(* Logix 5000 project; controller RSL5k_18_Template_noLib Emulate 5570 rev 32.11; software revision 32.02; part 4 of 16 *)
(* tags used below, declared in another part *)
   Cfg_AllowDisable : BOOL;   // 1=Allow Maintenance to Disable this Alarm
   PCmd_Reset : BOOL;   // Program Command to Reset latched alarm
   PCmd_Ack : BOOL;   // Program Command to Acknowledge alarm
   PCmd_Suppress : BOOL;   // Program Command to Suppress by Design (inhibits new alarm)
   PCmd_Unsuppress : BOOL;   // Program Command to Unsuppress (allows new alarm)
   PCmd_Unshelve : BOOL;   // Program Command to Unshelve (e.g., on shift change)
   Shelved : ALIAS FOR Com_AE.3;   // 1=Alarm has been Shelved by Operator (inhibits new alarm)
   Suppressed : ALIAS FOR Com_AE.6;   // 1=Alarm has been Suppressed by Program (inhibits new alarm)
   Disabled : ALIAS FOR Com_AE.9;   // 1=Alarm has been Disabled by Maintanance (inhibits new alarm)
   P_Alarm : BOOL;   // Unique Parameter Name for auto - discovery
   Wrk_Suppressed : BOOL;   // Internal Alarm Suppressed Status
   Com_AE : INT;   // Communication with HMI / Alarm/Event Server (see bit descriptions)
   OCmd_Unshelve : BOOL;   // Operator Command to Unshelve alarm (allows new alarm)
   OCmd_Shelve : BOOL;   // Operator Command to Shelve Alarm (inhibits new alarm)
   OCmd_Ack : BOOL;   // Operator Command to Acknowledge alarm
   OCmd_Reset : BOOL;   // Operator Command to Reset latched alarm
   MCmd_Enable : BOOL;   // Maintenance Command to Enable alarm (allows new alarm)
   MCmd_Disable : BOOL;   // Maintenance Command to Disable alarm (inhibits new alarm)
(* P_Alarm, continued *)

ROUTINE Prescan   (* ladder *)
// Clear "lurking" Commands
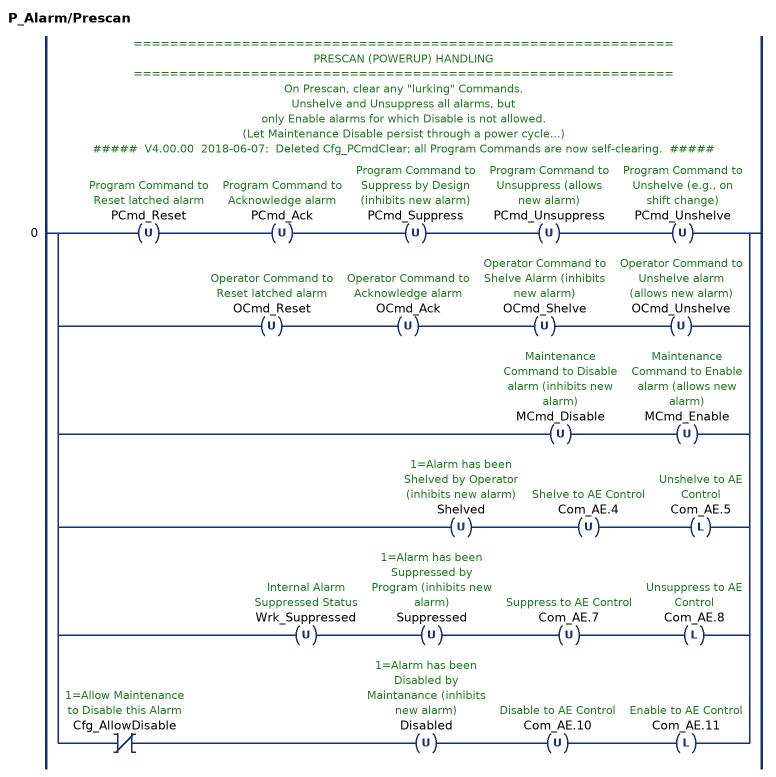
   // ============================================================
   // PRESCAN (POWERUP) HANDLING
   // ============================================================
   // On Prescan, clear any "lurking" Commands.
   // Unshelve and Unsuppress all alarms, but
   // only Enable alarms for which Disable is not allowed.
   // (Let Maintenance Disable persist through a power cycle...)
   // #####  V4.00.00  2018-06-07:  Deleted Cfg_PCmdClear; all Program Commands are now self-clearing.  #####
   0: [OTU(PCmd_Reset) OTU(PCmd_Ack) OTU(PCmd_Suppress) OTU(PCmd_Unsuppress) OTU(PCmd_Unshelve) ,OTU(OCmd_Reset) OTU(OCmd_Ack) OTU(OCmd_Shelve) OTU(OCmd_Unshelve) ,OTU(MCmd_Disable) OTU(MCmd_Enable) ,OTU(Shelved) OTU(Com_AE.4) OTL(Com_AE.5) ,OTU(Wrk_Suppressed) OTU(Suppressed) OTU(Com_AE.7) OTL(Com_AE.8) ,XIO(Cfg_AllowDisable) OTU(Disabled) OTU(Com_AE.10) OTL(Com_AE.11) ];
END_ROUTINE
END_ADD_ON_INSTRUCTION

ADD_ON_INSTRUCTION P_CmdSrc   (* revision 4.10 .01 Release, vendor Rockwell Automation, ExecutePrescan, ExecuteEnableInFalse *)
// Command Source
// Revision note:
// See Instruction Help for a summary of changes, and see 4.10 Release Notes for details.
// Help:
// Copyright © Rockwell Automation, Inc.  All Rights Reserved.
// This instruction provides selection of Command Source for a Device-
// level object  (from highest priority to lowest):
// * Not Initialized
// * Hand (hardwired control, not controllable from I/O)
// * POoS (Programmed Out of Service) (EnableIn is false)
// * MOoS (Maintenance Out of Service)
// * Maint (Maintenance)
// * Ovrd (Override) (typically used for process overrides)
// * External (e.g.: local/field devices or upstream SCADA)
// * Prog (Program) (automated control, and default if Cfg_ProgDefault = 1)
// * Oper (Operator (manual control, and default if Cfg_ProgDefault = 0)
// (Program and Operator have the same priority.)
// The current command source is shown with individual Status bits
// and also a bit field (Sts_bSrc) and an enumeration (Sts_eSrc).
// When EnableIn is false, all source acquire/release and lock/unlock
// Commands are processed "behind the scenes", but the source
// "Program Out of Service" (POoS) is selected.  When EnableIn
// becomes true, the source selection takes into account the
// Commands received -- in other words, the command source
// becomes the one that would have been in effect had the EnableIn
// False / Out of Service condition never occurred.
// SUMMARY OF CHANGES FROM PREVIOUS VERSION (4.10.00)
// See 4.10 Release Notes for details.
// * Added clear of internal "Ext" latch if Ext does not exist.
// SUMMARY OF CHANGES FROM PREVIOUS VERSION (4.00.01)
// See 4.10 Release Notes for details.
// * Added XCmd_Acq, XCmd_Rel, Cfg_ExtAcqAsLevel, removed Inp_Ext.
// * Added XRdy_Acq, XRdy_Rel so XCmd_Acq, XCmd_Rel can be used on HMI.
// * Corrected parameter external access.
// SUMMARY OF CHANGES FROM PREVIOUS VERSION (4.00.00)
// See 4.00 Release Notes for details.
// Minor change to initialization, handling of level commands in EnableInFalse.
// SUMMARY OF CHANGES FROM PREVIOUS VERSION (P_Mode V3.5-01)
// See 4.00 Release Notes for details.
// * Derived from P_Mode V3.5-01. P_Mode version history archived.
// * Added Out of Service (OoS), External (Ext); removed "NoMode"
// * Added configuration for sources to exist, commands for "opposite" source.
// * Aligned ready bit naming with command bit names.
VAR_INPUT
   Inp_Hand : BOOL; {visible}   // 1=Acquire Hand (typ. hardwired local), 0=Release Hand
   Inp_Ovrd : BOOL; {visible}   // 1=Acquire Override (higher priority program logic), 0=Release Override
   Inp_ExtInh : BOOL; {visible}   // 1=Inhibit External Acquisition, 0=Allow External Acquisition
   Cfg_HasOper : BOOL := 1;   // 1=Operator (unlocked) exists, can be selected
   Cfg_HasOperLocked : BOOL := 1;   // 1=Operator Locked exists, can be selected
   Cfg_HasProg : BOOL := 1;   // 1=Program (unlocked) exists, can be selected
   Cfg_HasProgLocked : BOOL := 1;   // 1=Program Locked exists, can be selected
   Cfg_HasExt : BOOL;   // 1=External exists, can be selected
   Cfg_HasMaint : BOOL := 1;   // 1=Maintenance exists, can be selected
   Cfg_HasMOoS : BOOL := 1;   // 1=Maintenance Out of Service exists, can be selected
   Cfg_OvrdOverLock : BOOL := 1;   // 1=Override supersedes Prog/Oper Lock, 0=don't override Lock
   Cfg_ExtOverLock : BOOL;   // 1=External supersedes Prog/Oper Lock, 0=don't override Lock
   Cfg_ProgPwrUp : BOOL;   // 1=Power Up to Prog, 0=Power Up to Oper
   Cfg_ProgNormal : BOOL;   // Normal Source: 1=Program if no requests; 0=Operator if no requests
   Cfg_PCmdPriority : BOOL;   // Command Priority: 1=Program Cmds Win; 0=Operator Cmds Win
   Cfg_PCmdProgAsLevel : BOOL;   // 1=PCmd_Prog used as a Level (1=Prog, 0=Oper)
   Cfg_PCmdLockAsLevel : BOOL;   // 1=PCmd_Lock used as a Level (1=Lock, 0=Unlock)
   Cfg_ExtAcqAsLevel : BOOL;   // 1=XCmd_Acq used as Level (1=Acq, 0=Rel)
   PCmd_Oper : BOOL;   // Program Command to select Operator (Prog to Oper)
   PCmd_Prog : BOOL;   // Program Command to select Program (Oper to Prog)
   PCmd_Lock : BOOL;   // Program Command to Lock Program (disallow Operator)
   PCmd_Unlock : BOOL;   // Program Command to Unlock Program (allow Oper to acquire)
   PCmd_Normal : BOOL;   // Program Command to select Normal (Oper or Prog)
   MCmd_OoS : BOOL;   // Maintenance Command to select Out Of Service
   MCmd_IS : BOOL;   // Maintenance Command to select In Service
   MCmd_Acq : BOOL;   // Maintenance Command to Acquire (Oper/Prog/Ovrd to Maint)
   MCmd_Rel : BOOL;   // Maintenance Command to Release (Maint to Oper/Prog/Ovrd)
   XCmd_Acq : BOOL;   // External Command to Acquire
   XCmd_Rel : BOOL;   // External Command to Release
   OCmd_Oper : BOOL;   // Operator Command to select Operator (Prog to Oper)
   OCmd_Prog : BOOL;   // Operator Command to select Program (Oper to Prog)
   OCmd_Lock : BOOL;   // Operator Command to Lock Operator (disallow Program)
   OCmd_Unlock : BOOL;   // Operator Command to Unlock Operator (allow Prog to acquire)
   OCmd_Normal : BOOL;   // Operator Command to select Normal (Oper or Prog)
END_VAR
VAR_OUTPUT
   Sts_eSrc : INT; {access Read Only}   // Selection enum: .8=Ext, .7=OoS, .6=Oper, .5=Prog, .4=Ovrd, .3=Maint, .2=Hand, .1=Norm, .0=Lock
   Sts_bSrc : INT; {access Read Only}   // Active Selection bitmap (for HMI totem pole)
        .0   // Hand
        .1   // Programmable Out of Service
        .2   // Maintenance Out of Service
        .3   // Maintenance
        .4   // Override
        .5   // External
        .6   // Program Locked
        .7   // Program
        .8   // Operator Locked
        .9   // Operator
   Sts_Hand : BOOL; {access Read Only, visible}   // 1=Hand is selected (supersedes OoS, Maint, Ovrd, Ext, Prog, Oper)
   Sts_OoS : BOOL; {access Read Only, visible}   // 1=Out of Service is selected (supersedes Maint, Ovrd, Ext, Prog, Oper)
   Sts_Maint : BOOL; {access Read Only, visible}   // 1=Maintenance is selected (supersedes Ovrd, Ext, Prog, Oper)
   Sts_Ovrd : BOOL; {access Read Only, visible}   // 1=Override is selected (supersedes Ext, Prog, Oper)
   Sts_Ext : BOOL; {access Read Only, visible}   // 1=External is selected (supersedes Prog, Oper)
   Sts_Prog : BOOL; {access Read Only, visible}   // 1=Program is selected
   Sts_ProgLocked : BOOL; {access Read Only}   // 1=Program is selected and Locked
   Sts_Oper : BOOL; {access Read Only, visible}   // 1=Operator is selected
   Sts_OperLocked : BOOL; {access Read Only}   // 1=Operator is selected and Locked
   Sts_ProgOperSel : BOOL; {access Read Only}   // Prog/Oper selection (latch) state, 1=Program, 0=Operator
   Sts_ProgOperLock : BOOL; {access Read Only, visible}   // Prog/Oper lock (latch) state, 1=Locked, 0=Unlocked
   Sts_Normal : BOOL; {access Read Only}   // 1=Selection equals the Normal (Prog or Oper)
   Sts_ProgReqInh : BOOL; {access Read Only}   // 1=Program request inhibited, cannot Get to Program from Current State
   Sts_ExtReqInh : BOOL; {access Read Only}   // 1=External request inhibited
   Sts_MAcqRcvd : BOOL; {access Read Only}   // 1=Maintenance Acquire command received this scan
   MRdy_OoS : BOOL; {access Read Only}   // 1=Ready for MCmd_OoS (enables HMI button)
   MRdy_IS : BOOL; {access Read Only}   // 1=Ready for MCmd_IS (enables HMI button)
   MRdy_Acq : BOOL; {access Read Only}   // 1=Ready for MCmd_Acq (enables HMI button)
   MRdy_Rel : BOOL; {access Read Only}   // 1=Ready for MCmd_Rel (enables HMI button)
   XRdy_Acq : BOOL; {access Read Only}   // 1=Ready for XCmd_Acq (enables HMI button)
   XRdy_Rel : BOOL; {access Read Only}   // 1=Ready for XCmd_Rel (enables HMI button)
   ORdy_Oper : BOOL; {access Read Only}   // 1=Ready for OCmd_Oper (enables HMI button)
   ORdy_Prog : BOOL; {access Read Only}   // 1=Ready for OCmd_Prog (enables HMI button)
   ORdy_Lock : BOOL; {access Read Only}   // 1=Ready for OCmd_Lock (enables HMI button)
   ORdy_Unlock : BOOL; {access Read Only}   // 1=Ready for OCmd_Unlock (enables HMI button)
   ORdy_Normal : BOOL; {access Read Only}   // 1=Ready for OCmd_Normal (enables HMI button)
   P_CmdSrc : BOOL;   // Unique Parameter Name for auto - discovery
END_VAR
VAR
   Wrk_ProgOperSel : BOOL; {access None}   // Internal Program (1) / Operator (0) selection result
   Wrk_ProgOperLock : BOOL; {access None}   // Internal Prog/Oper Lock (1) / Unlock (0) selection result
   Wrk_Prog : BOOL; {access None}   // Internal Program (1) / Operator (0) selection progress
   Wrk_MOoS : BOOL; {access None}   // Internal Maintenance Out of Service (1) / In Service (0) latch
   Wrk_Maint : BOOL; {access None}   // Internal Maintenance Acquire (1) / Release (0) latch
   Wrk_Lock : BOOL; {access None}   // Internal Prog/Oper Lock (1) / Unlock (0) selection progress
   Wrk_Init : BOOL; {access None}   // 1=Initialized, 0=Initialization is required (e.g., powerup)
   Wrk_HasProgLocked : BOOL; {access None}   // Stored copy of Cfg_HasProgLocked
   Wrk_HasProg : BOOL; {access None}   // Stored copy of Cfg_HasProg
   Wrk_HasOperLocked : BOOL; {access None}   // Stored copy of Cfg_HasOperLocked
   Wrk_HasOper : BOOL; {access None}   // Stored copy of Cfg_HasOper
   HMI_Type : STRING_12 := 'P_CmdSrc'; {access Read Only}   // Must contain AOI name, used for HMI and Information S/W
   HMI_Lib : STRING_8 := 'RA-BAS'; {access Read Only}   // Display Library for Faceplate call-up
   Wrk_Ext : BOOL; {access None}   // Internal latch of External selection (1=Ext acquired)
END_VAR

ROUTINE EnableInFalse   (* ladder *)
// Processes received Commands, but shows "Programmed Out of Service"
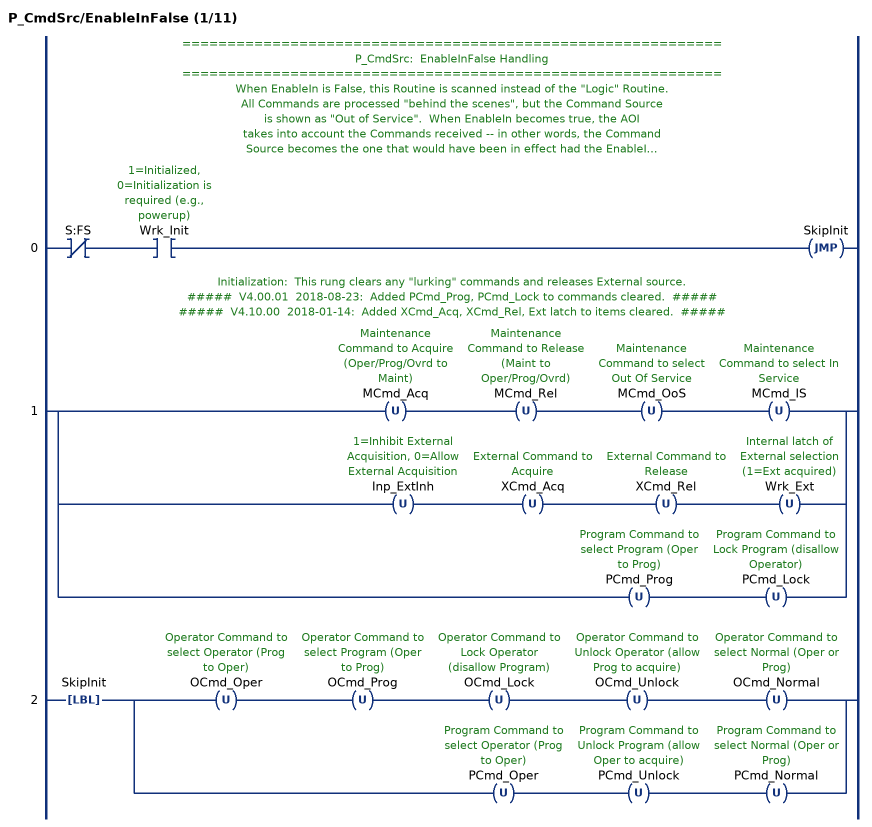
   // ============================================================
   // P_CmdSrc:  EnableInFalse Handling
   // ============================================================
   // When EnableIn is False, this Routine is scanned instead of the "Logic" Routine.
   // All Commands are processed "behind the scenes", but the Command Source
   // is shown as "Out of Service".  When EnableIn becomes true, the AOI
   // takes into account the Commands received -- in other words, the Command
   // Source becomes the one that would have been in effect had the EnableIn
   // False / Out of Service condition never occurred.
   // ============================================================
   // INITIALIZATION
   // ============================================================
   // If initialization has been completed, skip the following few rungs.
   0: XIO(S:FS)XIC(Wrk_Init)JMP(SkipInit);
   // Initialization:  This rung clears any "lurking" commands and releases External source.
   // #####  V4.00.01  2018-08-23:  Added PCmd_Prog, PCmd_Lock to commands cleared.  #####
   // #####  V4.10.00  2018-01-14:  Added XCmd_Acq, XCmd_Rel, Ext latch to items cleared.  #####
   1: [OTU(MCmd_Acq) OTU(MCmd_Rel) OTU(MCmd_OoS) OTU(MCmd_IS) ,OTU(Inp_ExtInh) OTU(XCmd_Acq) OTU(XCmd_Rel) OTU(Wrk_Ext) ,OTU(PCmd_Prog) OTU(PCmd_Lock) ];
   2: LBL(SkipInit)[OTU(OCmd_Oper) OTU(OCmd_Prog) OTU(OCmd_Lock) OTU(OCmd_Unlock) OTU(OCmd_Normal) ,OTU(PCmd_Oper) OTU(PCmd_Unlock) OTU(PCmd_Normal) ];
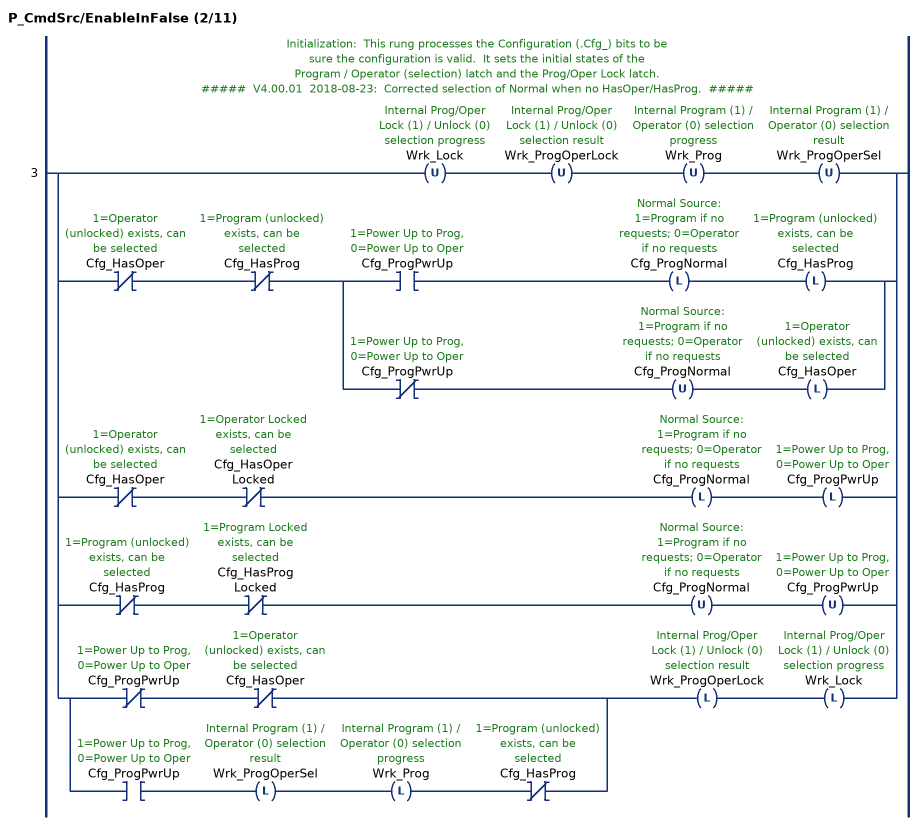
   // Initialization:  This rung processes the Configuration (.Cfg_) bits to be
   // sure the configuration is valid.  It sets the initial states of the
   // Program / Operator (selection) latch and the Prog/Oper Lock latch.
   // #####  V4.00.01  2018-08-23:  Corrected selection of Normal when no HasOper/HasProg.  #####
   3: [OTU(Wrk_Lock) OTU(Wrk_ProgOperLock) OTU(Wrk_Prog) OTU(Wrk_ProgOperSel) ,XIO(Cfg_HasOper) XIO(Cfg_HasProg) [XIC(Cfg_ProgPwrUp) OTL(Cfg_ProgNormal) OTL(Cfg_HasProg) ,XIO(Cfg_ProgPwrUp) OTU(Cfg_ProgNormal) OTL(Cfg_HasOper) ] ,XIO(Cfg_HasOper) XIO(Cfg_HasOperLocked) OTL(Cfg_ProgNormal) OTL(Cfg_ProgPwrUp) ,XIO(Cfg_HasProg) XIO(Cfg_HasProgLocked) OTU(Cfg_ProgNormal) OTU(Cfg_ProgPwrUp) ,[XIO(Cfg_ProgPwrUp) XIO(Cfg_HasOper) ,XIC(Cfg_ProgPwrUp) OTL(Wrk_ProgOperSel) OTL(Wrk_Prog) XIO(Cfg_HasProg) ] OTL(Wrk_ProgOperLock) OTL(Wrk_Lock) ];
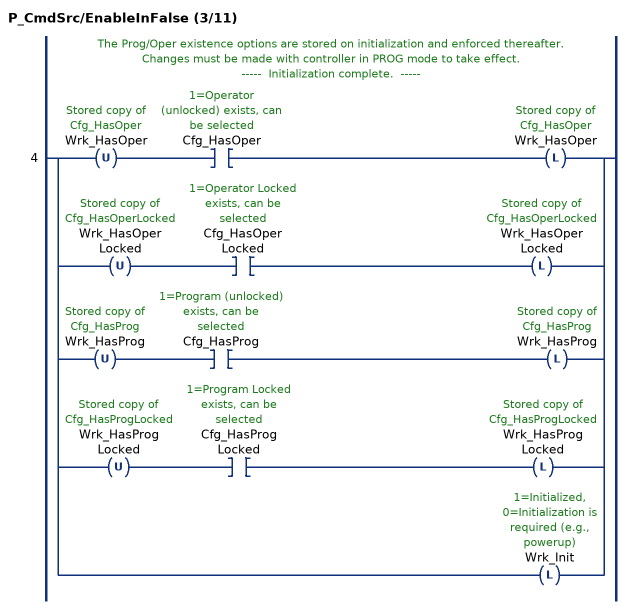
   // The Prog/Oper existence options are stored on initialization and enforced thereafter.
   // Changes must be made with controller in PROG mode to take effect.
   // -----  Initialization complete.  -----
   4: [OTU(Wrk_HasOper) XIC(Cfg_HasOper) OTL(Wrk_HasOper) ,OTU(Wrk_HasOperLocked) XIC(Cfg_HasOperLocked) OTL(Wrk_HasOperLocked) ,OTU(Wrk_HasProg) XIC(Cfg_HasProg) OTL(Wrk_HasProg) ,OTU(Wrk_HasProgLocked) XIC(Cfg_HasProgLocked) OTL(Wrk_HasProgLocked) ,OTL(Wrk_Init) ];
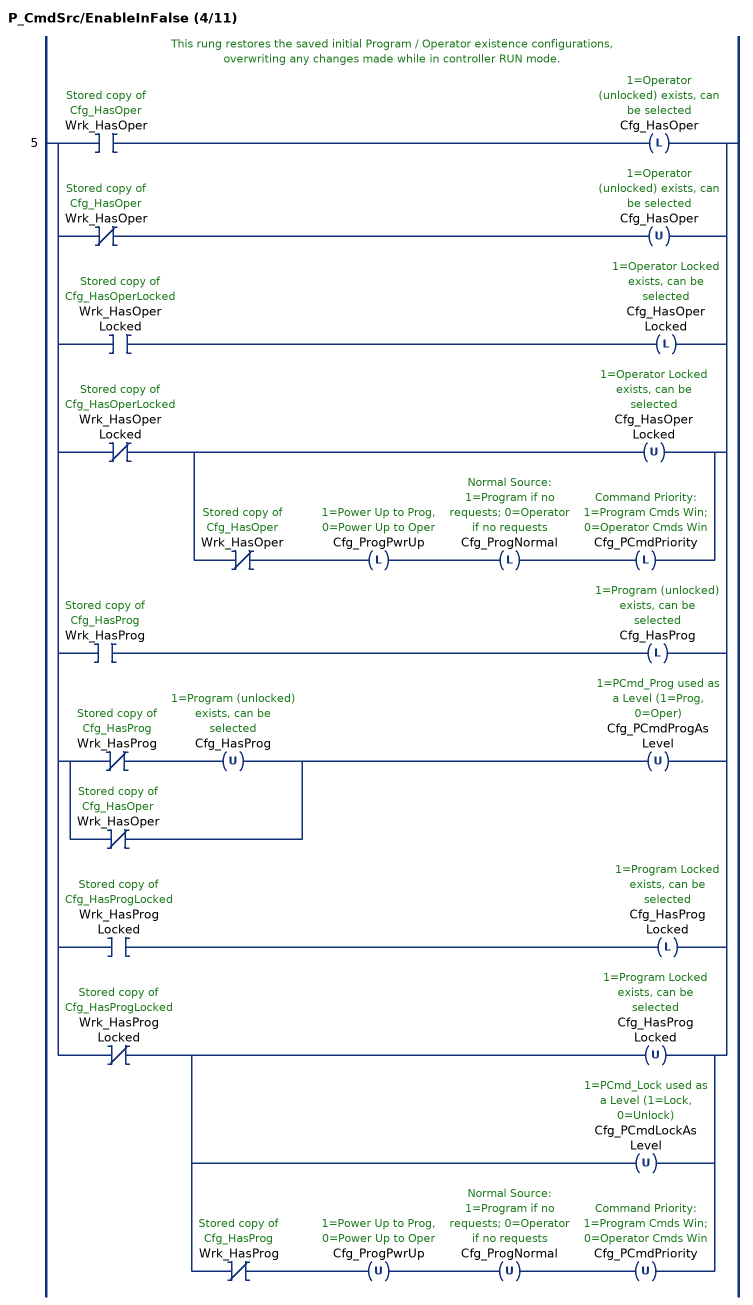
   // This rung restores the saved initial Program / Operator existence configurations,
   // overwriting any changes made while in controller RUN mode.
   5: [XIC(Wrk_HasOper) OTL(Cfg_HasOper) ,XIO(Wrk_HasOper) OTU(Cfg_HasOper) ,XIC(Wrk_HasOperLocked) OTL(Cfg_HasOperLocked) ,XIO(Wrk_HasOperLocked) [OTU(Cfg_HasOperLocked) ,XIO(Wrk_HasOper) OTL(Cfg_ProgPwrUp) OTL(Cfg_ProgNormal) OTL(Cfg_PCmdPriority) ] ,XIC(Wrk_HasProg) OTL(Cfg_HasProg) ,[XIO(Wrk_HasProg) OTU(Cfg_HasProg) ,XIO(Wrk_HasOper) ] OTU(Cfg_PCmdProgAsLevel) ,XIC(Wrk_HasProgLocked) OTL(Cfg_HasProgLocked) ,XIO(Wrk_HasProgLocked) [[OTU(Cfg_HasProgLocked) ,OTU(Cfg_PCmdLockAsLevel) ] ,XIO(Wrk_HasProg) OTU(Cfg_ProgPwrUp) OTU(Cfg_ProgNormal) OTU(Cfg_PCmdPriority) ] ];
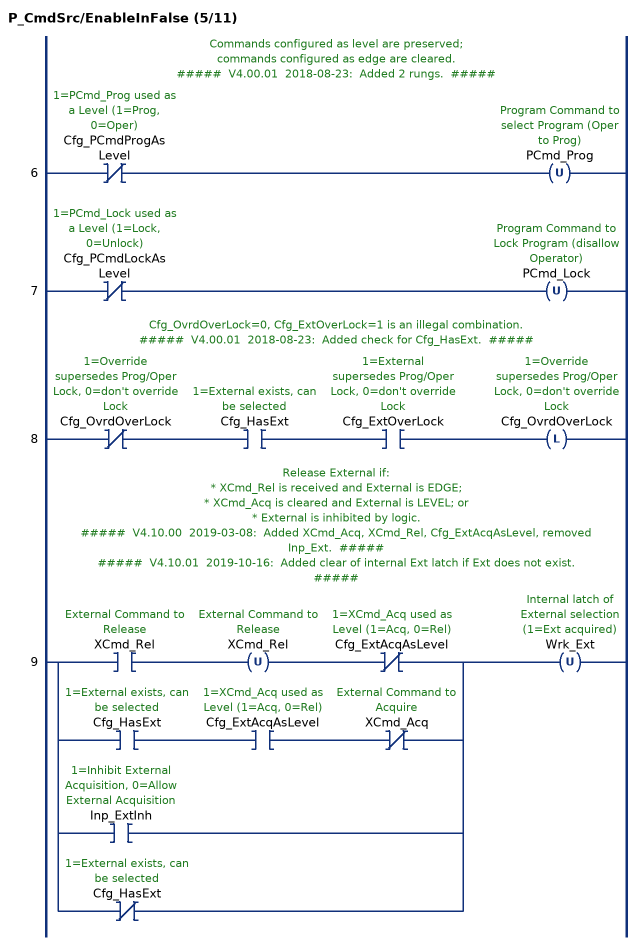
   // Commands configured as level are preserved;
   // commands configured as edge are cleared.
   // #####  V4.00.01  2018-08-23:  Added 2 rungs.  #####
   6: XIO(Cfg_PCmdProgAsLevel)OTU(PCmd_Prog);
   7: XIO(Cfg_PCmdLockAsLevel)OTU(PCmd_Lock);
   // Cfg_OvrdOverLock=0, Cfg_ExtOverLock=1 is an illegal combination.
   // #####  V4.00.01  2018-08-23:  Added check for Cfg_HasExt.  #####
   8: XIO(Cfg_OvrdOverLock)XIC(Cfg_HasExt)XIC(Cfg_ExtOverLock)OTL(Cfg_OvrdOverLock);
   // Release External if:
   // * XCmd_Rel is received and External is EDGE;
   // * XCmd_Acq is cleared and External is LEVEL; or
   // * External is inhibited by logic.
   // #####  V4.10.00  2019-03-08:  Added XCmd_Acq, XCmd_Rel, Cfg_ExtAcqAsLevel, removed Inp_Ext.  #####
   // #####  V4.10.01  2019-10-16:  Added clear of internal Ext latch if Ext does not exist.  #####
   9: [XIC(XCmd_Rel) OTU(XCmd_Rel) XIO(Cfg_ExtAcqAsLevel) ,XIC(Cfg_HasExt) XIC(Cfg_ExtAcqAsLevel) XIO(XCmd_Acq) ,XIC(Inp_ExtInh) ,XIO(Cfg_HasExt) ]OTU(Wrk_Ext);
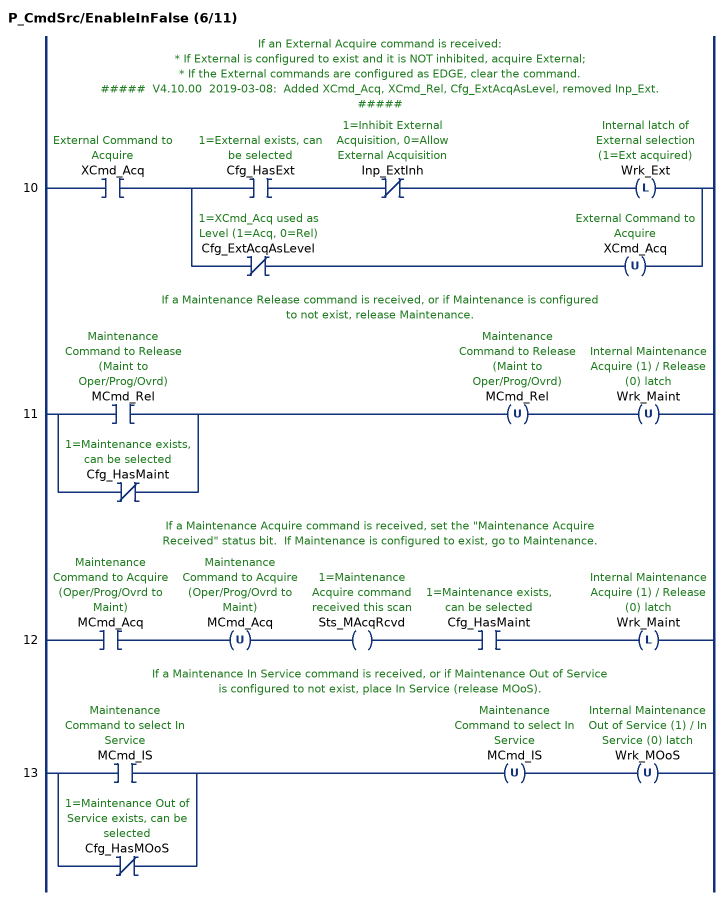
   // If an External Acquire command is received:
   // * If External is configured to exist and it is NOT inhibited, acquire External;
   // * If the External commands are configured as EDGE, clear the command.
   // #####  V4.10.00  2019-03-08:  Added XCmd_Acq, XCmd_Rel, Cfg_ExtAcqAsLevel, removed Inp_Ext.  #####
   10: XIC(XCmd_Acq)[XIC(Cfg_HasExt) XIO(Inp_ExtInh) OTL(Wrk_Ext) ,XIO(Cfg_ExtAcqAsLevel) OTU(XCmd_Acq) ];
   // If a Maintenance Release command is received, or if Maintenance is configured
   // to not exist, release Maintenance.
   11: [XIC(MCmd_Rel) ,XIO(Cfg_HasMaint) ]OTU(MCmd_Rel)OTU(Wrk_Maint);
   // If a Maintenance Acquire command is received, set the "Maintenance Acquire
   // Received" status bit.  If Maintenance is configured to exist, go to Maintenance.
   12: XIC(MCmd_Acq)OTU(MCmd_Acq)OTE(Sts_MAcqRcvd)XIC(Cfg_HasMaint)OTL(Wrk_Maint);
   // If a Maintenance In Service command is received, or if Maintenance Out of Service
   // is configured to not exist, place In Service (release MOoS).
   13: [XIC(MCmd_IS) ,XIO(Cfg_HasMOoS) ]OTU(MCmd_IS)OTU(Wrk_MOoS);
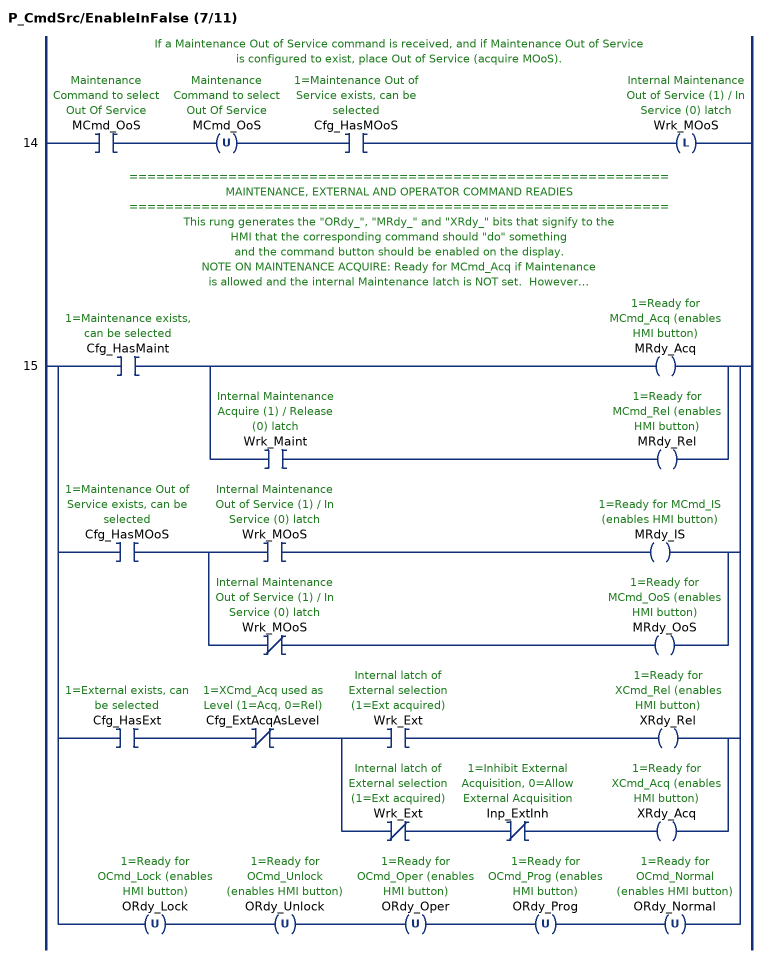
   // If a Maintenance Out of Service command is received, and if Maintenance Out of Service
   // is configured to exist, place Out of Service (acquire MOoS).
   14: XIC(MCmd_OoS)OTU(MCmd_OoS)XIC(Cfg_HasMOoS)OTL(Wrk_MOoS);
   // ============================================================
   // MAINTENANCE, EXTERNAL AND OPERATOR COMMAND READIES
   // ============================================================
   // This rung generates the "ORdy_", "MRdy_" and "XRdy_" bits that signify to the
   // HMI that the corresponding command should "do" something
   // and the command button should be enabled on the display.
   // NOTE ON MAINTENANCE ACQUIRE: Ready for MCmd_Acq if Maintenance
   // is allowed and the internal Maintenance latch is NOT set.  However,
   // we need to display Ready even if latch IS set so that Sts_MAcqRcvd
   // can blink to reset an external Maintenance expiration timer!!!
   // #####  V4.10.00  2019-03-08:  Added XRdy_Acq, XRdy_Rel so External Acq/Rel can be used on HMI .  #####
   15: [XIC(Cfg_HasMaint) [OTE(MRdy_Acq) ,XIC(Wrk_Maint) OTE(MRdy_Rel) ] ,XIC(Cfg_HasMOoS) [XIC(Wrk_MOoS) OTE(MRdy_IS) ,XIO(Wrk_MOoS) OTE(MRdy_OoS) ] ,XIC(Cfg_HasExt) XIO(Cfg_ExtAcqAsLevel) [XIC(Wrk_Ext) OTE(XRdy_Rel) ,XIO(Wrk_Ext) XIO(Inp_ExtInh) OTE(XRdy_Acq) ] ,OTU(ORdy_Lock) OTU(ORdy_Unlock) OTU(ORdy_Oper) OTU(ORdy_Prog) OTU(ORdy_Normal) ];
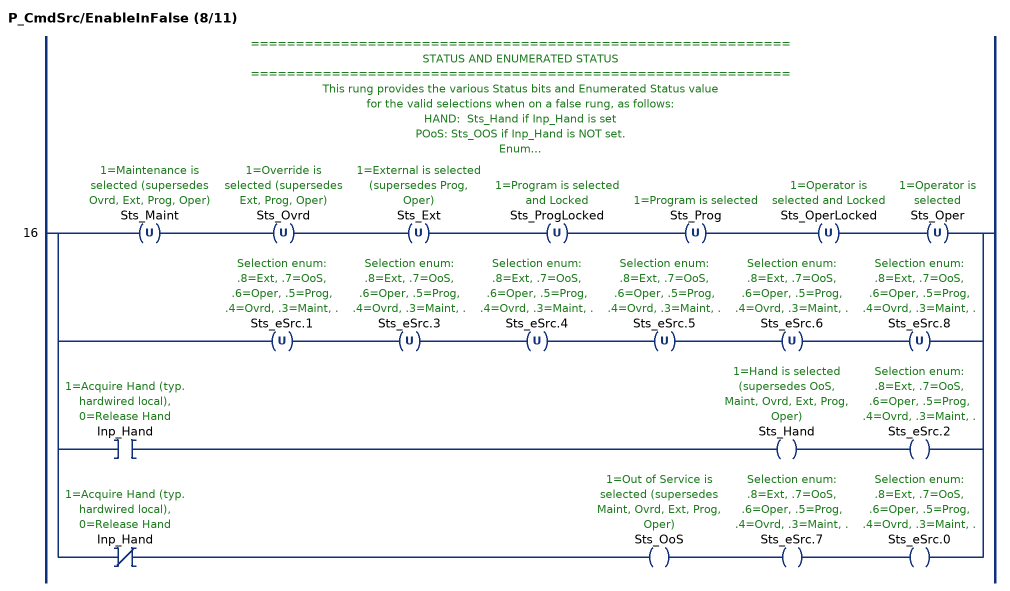
   // ============================================================
   // STATUS AND ENUMERATED STATUS
   // ============================================================
   // This rung provides the various Status bits and Enumerated Status value
   // for the valid selections when on a false rung, as follows:
   // HAND:  Sts_Hand if Inp_Hand is set
   // POoS: Sts_OOS if Inp_Hand is NOT set.
   // Enum:
   // = 4  if HAND
   // = 129 if POoS
   16: [OTU(Sts_Maint) OTU(Sts_Ovrd) OTU(Sts_Ext) OTU(Sts_ProgLocked) OTU(Sts_Prog) OTU(Sts_OperLocked) OTU(Sts_Oper) ,OTU(Sts_eSrc.1) OTU(Sts_eSrc.3) OTU(Sts_eSrc.4) OTU(Sts_eSrc.5) OTU(Sts_eSrc.6) OTU(Sts_eSrc.8) ,XIC(Inp_Hand) OTE(Sts_Hand) OTE(Sts_eSrc.2) ,XIO(Inp_Hand) OTE(Sts_OoS) OTE(Sts_eSrc.7) OTE(Sts_eSrc.0) ];
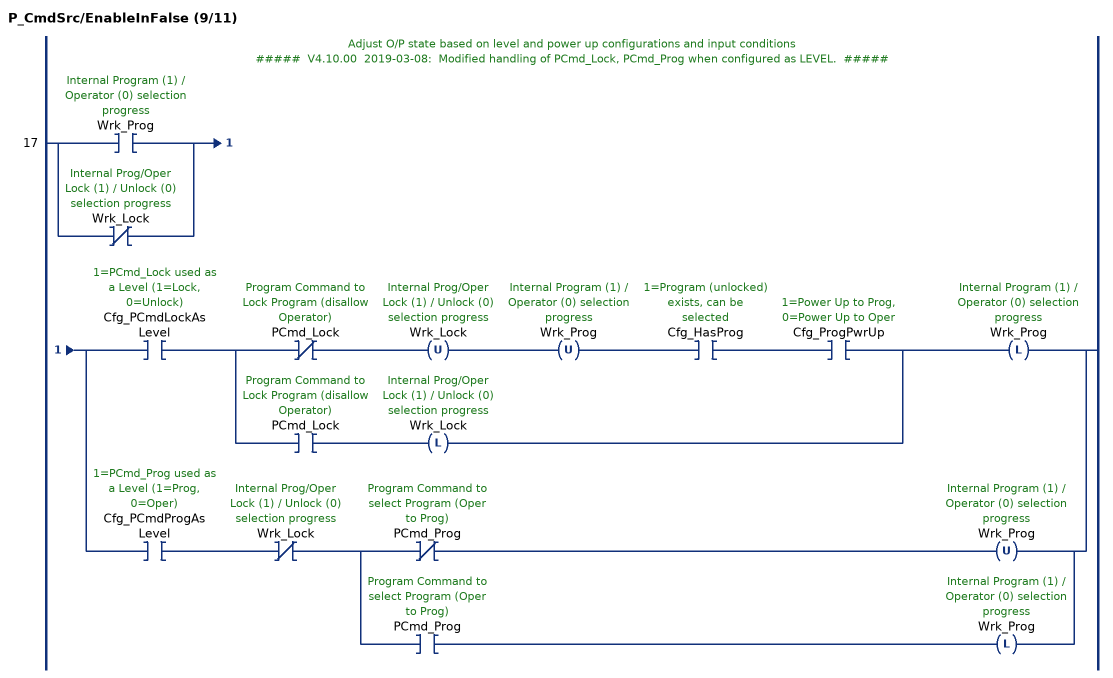
   // Adjust O/P state based on level and power up configurations and input conditions
   // #####  V4.10.00  2019-03-08:  Modified handling of PCmd_Lock, PCmd_Prog when configured as LEVEL.  #####
   17: [XIC(Wrk_Prog) ,XIO(Wrk_Lock) ][XIC(Cfg_PCmdLockAsLevel) [XIO(PCmd_Lock) OTU(Wrk_Lock) OTU(Wrk_Prog) XIC(Cfg_HasProg) XIC(Cfg_ProgPwrUp) ,XIC(PCmd_Lock) OTL(Wrk_Lock) ] OTL(Wrk_Prog) ,XIC(Cfg_PCmdProgAsLevel) XIO(Wrk_Lock) [XIO(PCmd_Prog) OTU(Wrk_Prog) ,XIC(PCmd_Prog) OTL(Wrk_Prog) ] ];
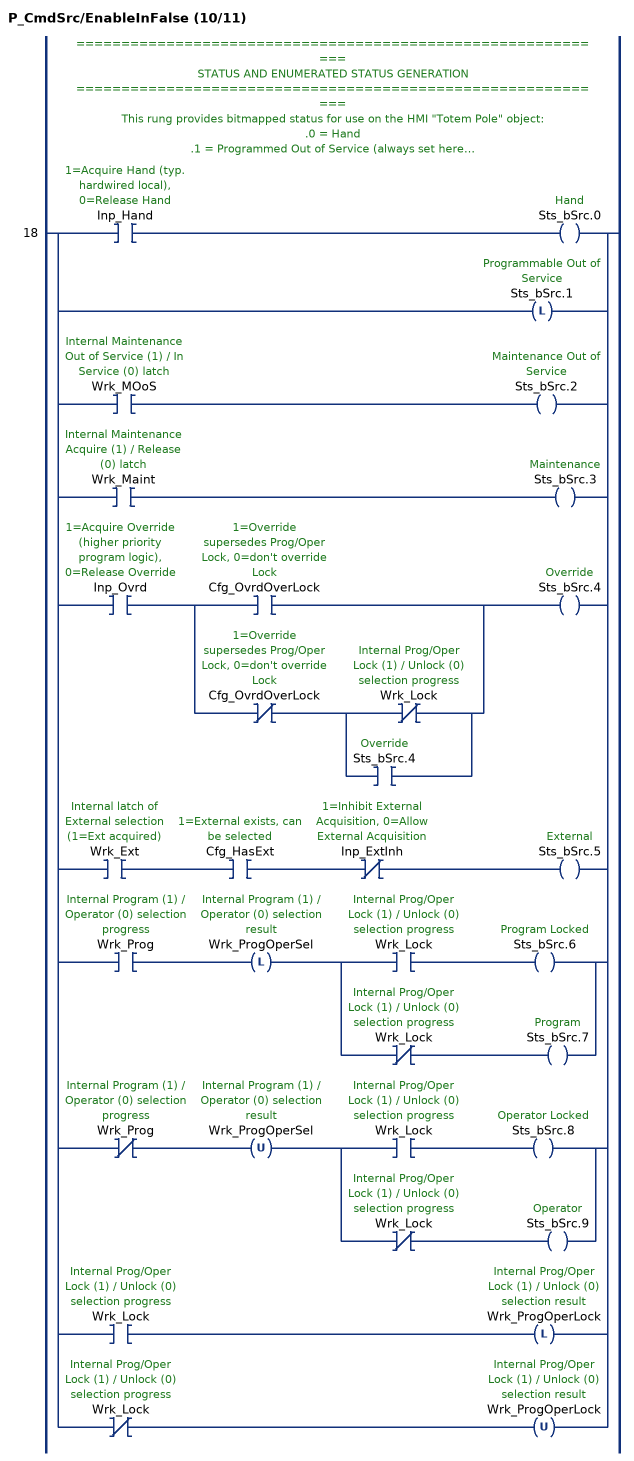
   // ============================================================
   // STATUS AND ENUMERATED STATUS GENERATION
   // ============================================================
   // This rung provides bitmapped status for use on the HMI "Totem Pole" object:
   // .0 = Hand
   // .1 = Programmed Out of Service (always set here)
   // .2 = Maintenance Out of Service
   // .3 = Maintenance
   // .4= Override
   // .5 = External
   // .6 = Program Locked
   // .7 = Program
   // .8 = Operator Locked
   // .9 = Operator
   // In addition, the final selections of the Program / Operator selection latch
   // and the Prog/Oper lock latch are captured for use next scan.
   // #####  V4.10.00  2019-03-08:  Added XCmd_Acq, XCmd_Rel, Cfg_ExtAcqAsLevel, removed Inp_Ext.  #####
   18: [XIC(Inp_Hand) OTE(Sts_bSrc.0) ,OTL(Sts_bSrc.1) ,XIC(Wrk_MOoS) OTE(Sts_bSrc.2) ,XIC(Wrk_Maint) OTE(Sts_bSrc.3) ,XIC(Inp_Ovrd) [XIC(Cfg_OvrdOverLock) ,XIO(Cfg_OvrdOverLock) [XIO(Wrk_Lock) ,XIC(Sts_bSrc.4) ] ] OTE(Sts_bSrc.4) ,XIC(Wrk_Ext) XIC(Cfg_HasExt) XIO(Inp_ExtInh) OTE(Sts_bSrc.5) ,XIC(Wrk_Prog) OTL(Wrk_ProgOperSel) [XIC(Wrk_Lock) OTE(Sts_bSrc.6) ,XIO(Wrk_Lock) OTE(Sts_bSrc.7) ] ,XIO(Wrk_Prog) OTU(Wrk_ProgOperSel) [XIC(Wrk_Lock) OTE(Sts_bSrc.8) ,XIO(Wrk_Lock) OTE(Sts_bSrc.9) ] ,XIC(Wrk_Lock) OTL(Wrk_ProgOperLock) ,XIO(Wrk_Lock) OTU(Wrk_ProgOperLock) ];
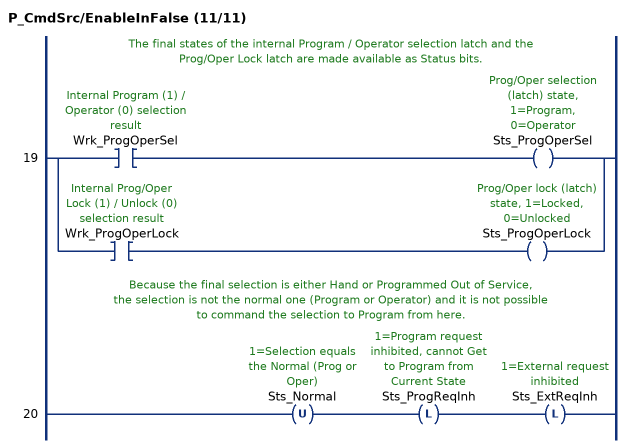
   // The final states of the internal Program / Operator selection latch and the
   // Prog/Oper Lock latch are made available as Status bits.
   19: [XIC(Wrk_ProgOperSel) OTE(Sts_ProgOperSel) ,XIC(Wrk_ProgOperLock) OTE(Sts_ProgOperLock) ];
   // Because the final selection is either Hand or Programmed Out of Service,
   // the selection is not the normal one (Program or Operator) and it is not possible
   // to command the selection to Program from here.
   20: OTU(Sts_Normal)OTL(Sts_ProgReqInh)OTL(Sts_ExtReqInh);
END_ROUTINE

ROUTINE Logic   (* ladder *)
// Selects Hand, OOS, Maint, Ovrd, Ext, Oper, Prog based on Inputs and Commands
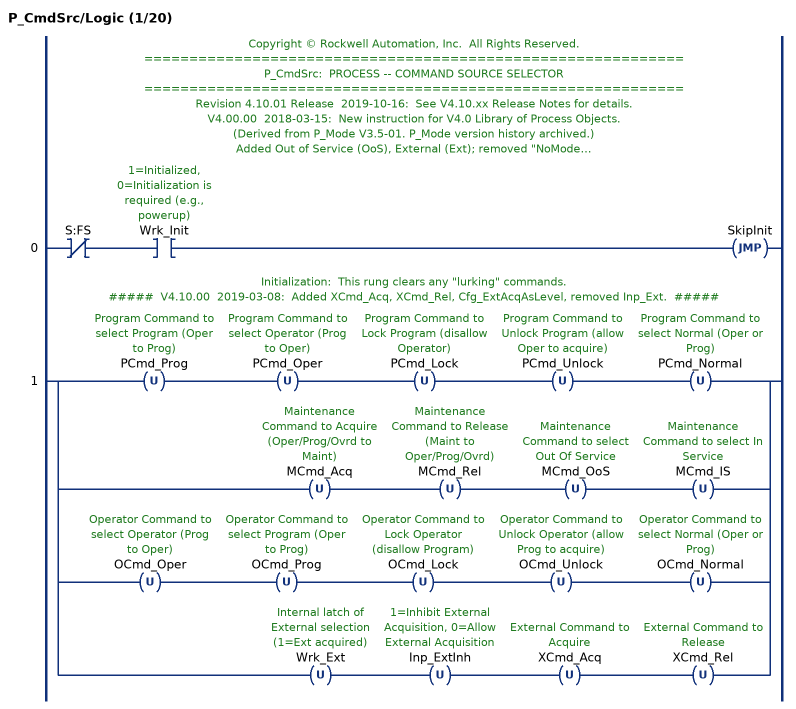
   // Copyright © Rockwell Automation, Inc.  All Rights Reserved.
   // ============================================================
   // P_CmdSrc:  PROCESS -- COMMAND SOURCE SELECTOR
   // ============================================================
   // Revision 4.10.01 Release  2019-10-16:  See V4.10.xx Release Notes for details.
   // V4.00.00  2018-03-15:  New instruction for V4.0 Library of Process Objects.
   // (Derived from P_Mode V3.5-01. P_Mode version history archived.)
   // Added Out of Service (OoS), External (Ext); removed "NoMode"
   // Added configuration for sources to exist, commands for "opposite" source.
   // Aligned ready bit naming with command bit names.
   // V4.00.01  2018-08-23:  Minor change to initialization, handling of level commands in EIF.
   // V4.10.00  2019-03-08:  Added XCmd_Acq, XCmd_Rel, Cfg_ExtAcqAsLevel, removed Inp_Ext.
   // Added XRdy_Acq, XRdy_Rel so XCmd_Acq, XCmd_Rel can be used on HMI.
   // Corrected parameter external access.
   // V4.10.01  2019-10-16:  Added clear of internal "Ext" latch if Ext does not exist.
   // ============================================================
   // This instruction provides selection of Command Source for a
   // Device-level object  (from highest priority to lowest):
   // * Not Initialized
   // * Hand (hardwired control, not controllable from I/O)
   // * POoS (programmed Out of Service) (EnableIn is false)
   // * MOoS (maintenance Out of Service)
   // * Maint (Maintenance)
   // *  Ovrd (Override) (typically used for process overrides)
   // * External (e.g.: field pilot controls or upstream SCADA)
   // *  Prog  (Program) (automated control, and default if Cfg_ProgNormal = 1)
   // *  Oper (Operator (manual control, and default if Cfg_ProgNormal = 0)
   // The current command source is shown with individual Status bits
   // and also a bit field (Sts_bSrc) and an enumeration (Sts_eSrc).
   // ============================================================
   // INITIALIZATION
   // ============================================================
   // If initialization has been completed, skip the following few rungs.
   0: XIO(S:FS)XIC(Wrk_Init)JMP(SkipInit);
   // Initialization:  This rung clears any "lurking" commands.
   // #####  V4.10.00  2019-03-08:  Added XCmd_Acq, XCmd_Rel, Cfg_ExtAcqAsLevel, removed Inp_Ext.  #####
   1: [OTU(PCmd_Prog) OTU(PCmd_Oper) OTU(PCmd_Lock) OTU(PCmd_Unlock) OTU(PCmd_Normal) ,OTU(MCmd_Acq) OTU(MCmd_Rel) OTU(MCmd_OoS) OTU(MCmd_IS) ,OTU(OCmd_Oper) OTU(OCmd_Prog) OTU(OCmd_Lock) OTU(OCmd_Unlock) OTU(OCmd_Normal) ,OTU(Wrk_Ext) OTU(Inp_ExtInh) OTU(XCmd_Acq) OTU(XCmd_Rel) ];
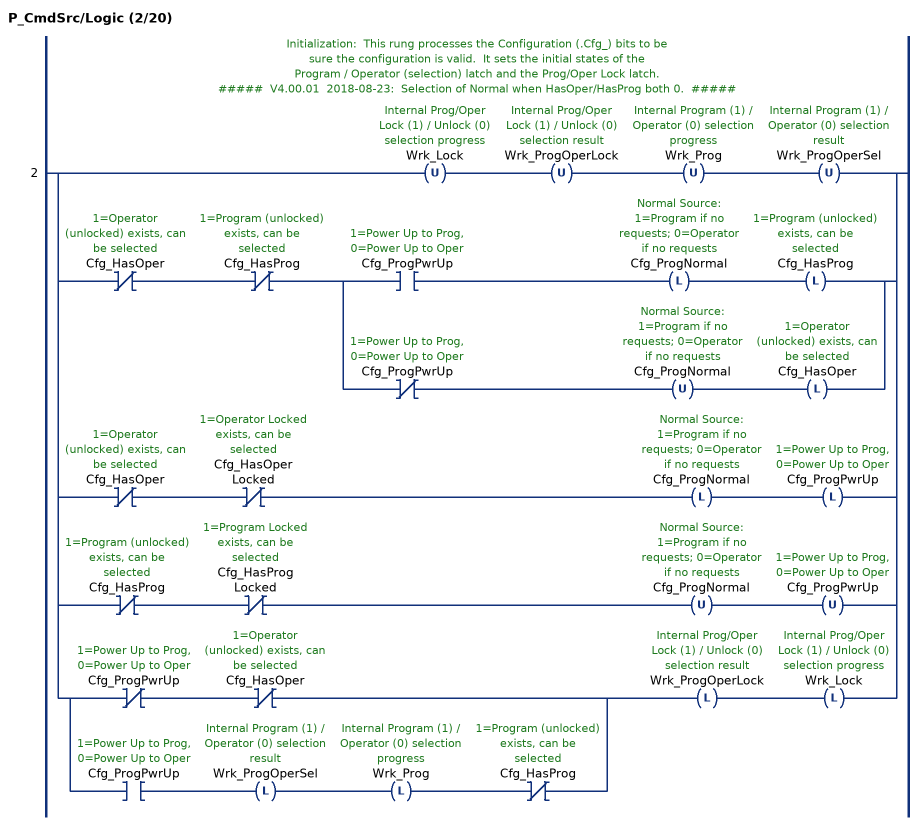
   // Initialization:  This rung processes the Configuration (.Cfg_) bits to be
   // sure the configuration is valid.  It sets the initial states of the
   // Program / Operator (selection) latch and the Prog/Oper Lock latch.
   // #####  V4.00.01  2018-08-23:  Selection of Normal when HasOper/HasProg both 0.  #####
   2: [OTU(Wrk_Lock) OTU(Wrk_ProgOperLock) OTU(Wrk_Prog) OTU(Wrk_ProgOperSel) ,XIO(Cfg_HasOper) XIO(Cfg_HasProg) [XIC(Cfg_ProgPwrUp) OTL(Cfg_ProgNormal) OTL(Cfg_HasProg) ,XIO(Cfg_ProgPwrUp) OTU(Cfg_ProgNormal) OTL(Cfg_HasOper) ] ,XIO(Cfg_HasOper) XIO(Cfg_HasOperLocked) OTL(Cfg_ProgNormal) OTL(Cfg_ProgPwrUp) ,XIO(Cfg_HasProg) XIO(Cfg_HasProgLocked) OTU(Cfg_ProgNormal) OTU(Cfg_ProgPwrUp) ,[XIO(Cfg_ProgPwrUp) XIO(Cfg_HasOper) ,XIC(Cfg_ProgPwrUp) OTL(Wrk_ProgOperSel) OTL(Wrk_Prog) XIO(Cfg_HasProg) ] OTL(Wrk_ProgOperLock) OTL(Wrk_Lock) ];
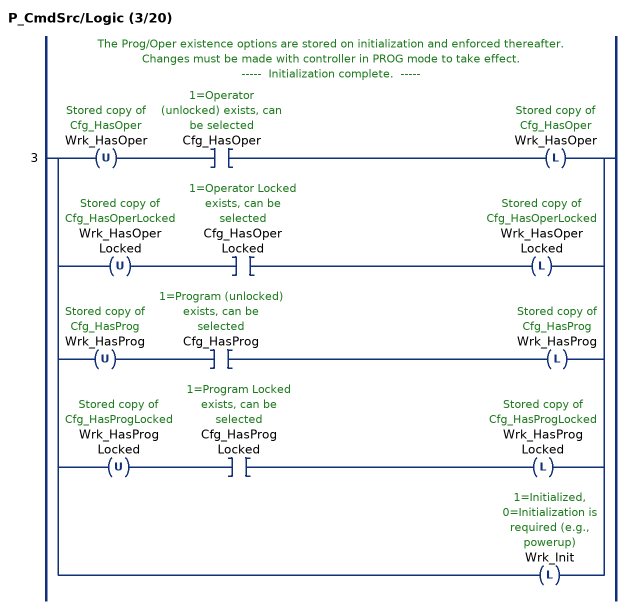
   // The Prog/Oper existence options are stored on initialization and enforced thereafter.
   // Changes must be made with controller in PROG mode to take effect.
   // -----  Initialization complete.  -----
   3: [OTU(Wrk_HasOper) XIC(Cfg_HasOper) OTL(Wrk_HasOper) ,OTU(Wrk_HasOperLocked) XIC(Cfg_HasOperLocked) OTL(Wrk_HasOperLocked) ,OTU(Wrk_HasProg) XIC(Cfg_HasProg) OTL(Wrk_HasProg) ,OTU(Wrk_HasProgLocked) XIC(Cfg_HasProgLocked) OTL(Wrk_HasProgLocked) ,OTL(Wrk_Init) ];
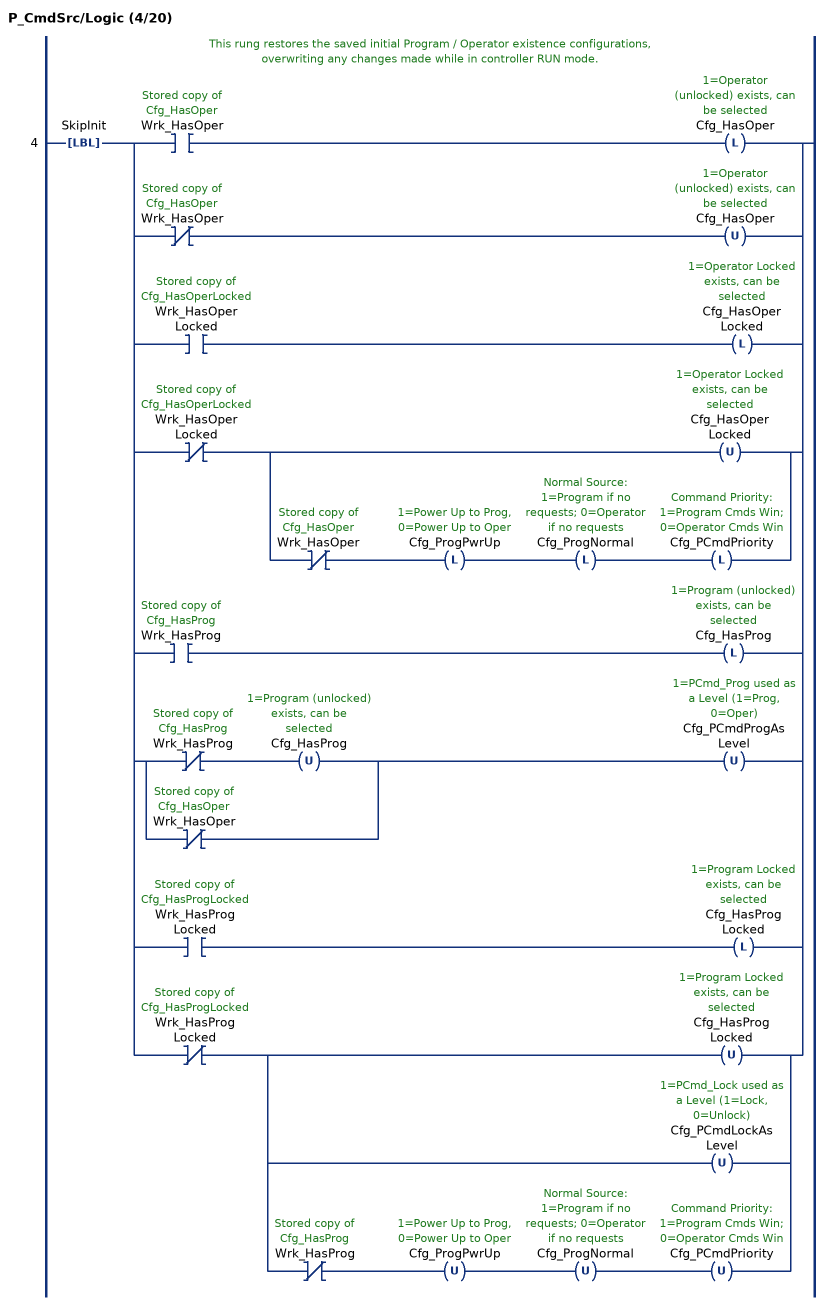
   // This rung restores the saved initial Program / Operator existence configurations,
   // overwriting any changes made while in controller RUN mode.
   4: LBL(SkipInit)[XIC(Wrk_HasOper) OTL(Cfg_HasOper) ,XIO(Wrk_HasOper) OTU(Cfg_HasOper) ,XIC(Wrk_HasOperLocked) OTL(Cfg_HasOperLocked) ,XIO(Wrk_HasOperLocked) [OTU(Cfg_HasOperLocked) ,XIO(Wrk_HasOper) OTL(Cfg_ProgPwrUp) OTL(Cfg_ProgNormal) OTL(Cfg_PCmdPriority) ] ,XIC(Wrk_HasProg) OTL(Cfg_HasProg) ,[XIO(Wrk_HasProg) OTU(Cfg_HasProg) ,XIO(Wrk_HasOper) ] OTU(Cfg_PCmdProgAsLevel) ,XIC(Wrk_HasProgLocked) OTL(Cfg_HasProgLocked) ,XIO(Wrk_HasProgLocked) [[OTU(Cfg_HasProgLocked) ,OTU(Cfg_PCmdLockAsLevel) ] ,XIO(Wrk_HasProg) OTU(Cfg_ProgPwrUp) OTU(Cfg_ProgNormal) OTU(Cfg_PCmdPriority) ] ];
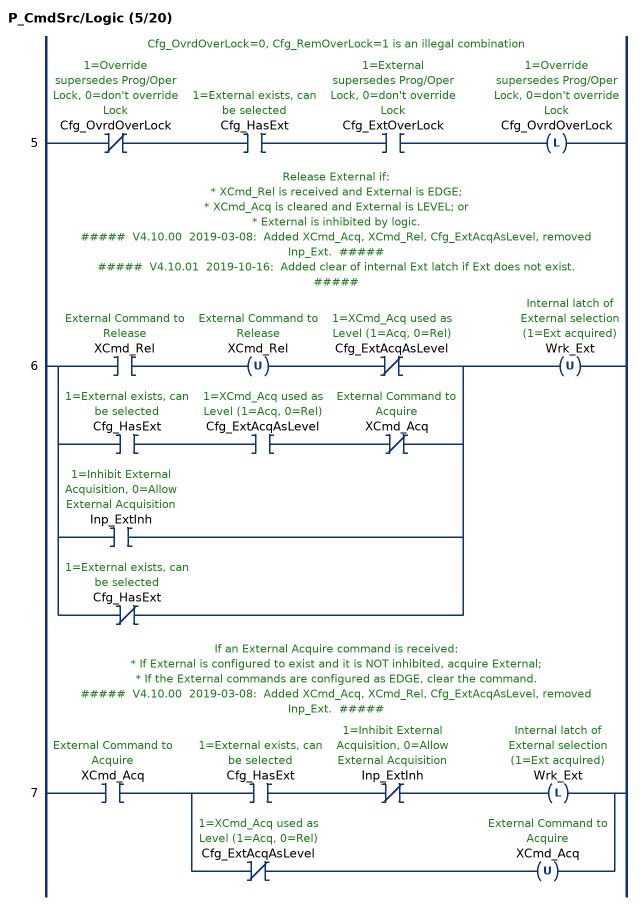
   // Cfg_OvrdOverLock=0, Cfg_RemOverLock=1 is an illegal combination
   5: XIO(Cfg_OvrdOverLock)XIC(Cfg_HasExt)XIC(Cfg_ExtOverLock)OTL(Cfg_OvrdOverLock);
   // Release External if:
   // * XCmd_Rel is received and External is EDGE;
   // * XCmd_Acq is cleared and External is LEVEL; or
   // * External is inhibited by logic.
   // #####  V4.10.00  2019-03-08:  Added XCmd_Acq, XCmd_Rel, Cfg_ExtAcqAsLevel, removed Inp_Ext.  #####
   // #####  V4.10.01  2019-10-16:  Added clear of internal Ext latch if Ext does not exist.  #####
   6: [XIC(XCmd_Rel) OTU(XCmd_Rel) XIO(Cfg_ExtAcqAsLevel) ,XIC(Cfg_HasExt) XIC(Cfg_ExtAcqAsLevel) XIO(XCmd_Acq) ,XIC(Inp_ExtInh) ,XIO(Cfg_HasExt) ]OTU(Wrk_Ext);
   // If an External Acquire command is received:
   // * If External is configured to exist and it is NOT inhibited, acquire External;
   // * If the External commands are configured as EDGE, clear the command.
   // #####  V4.10.00  2019-03-08:  Added XCmd_Acq, XCmd_Rel, Cfg_ExtAcqAsLevel, removed Inp_Ext.  #####
   7: XIC(XCmd_Acq)[XIC(Cfg_HasExt) XIO(Inp_ExtInh) OTL(Wrk_Ext) ,XIO(Cfg_ExtAcqAsLevel) OTU(XCmd_Acq) ];
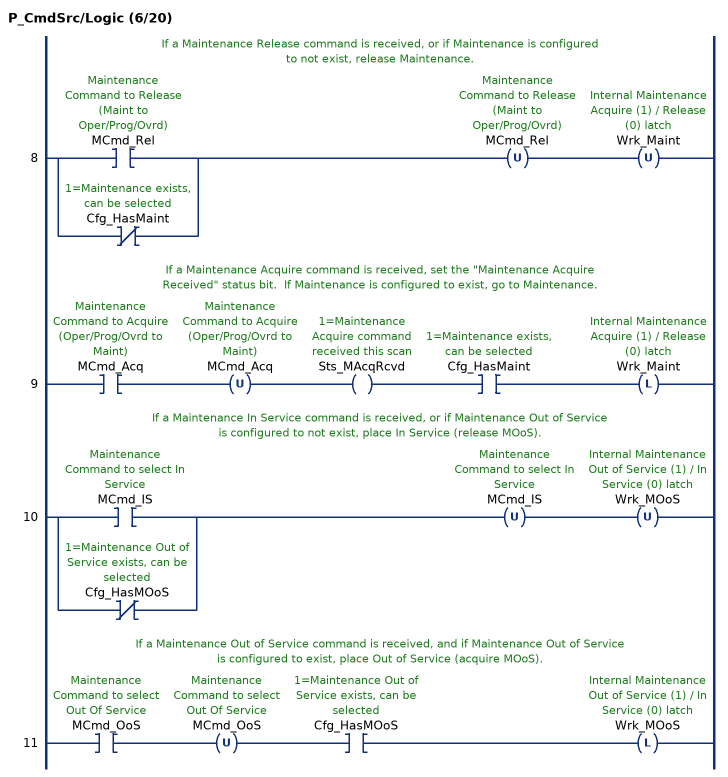
   // If a Maintenance Release command is received, or if Maintenance is configured
   // to not exist, release Maintenance.
   8: [XIC(MCmd_Rel) ,XIO(Cfg_HasMaint) ]OTU(MCmd_Rel)OTU(Wrk_Maint);
   // If a Maintenance Acquire command is received, set the "Maintenance Acquire
   // Received" status bit.  If Maintenance is configured to exist, go to Maintenance.
   9: XIC(MCmd_Acq)OTU(MCmd_Acq)OTE(Sts_MAcqRcvd)XIC(Cfg_HasMaint)OTL(Wrk_Maint);
   // If a Maintenance In Service command is received, or if Maintenance Out of Service
   // is configured to not exist, place In Service (release MOoS).
   10: [XIC(MCmd_IS) ,XIO(Cfg_HasMOoS) ]OTU(MCmd_IS)OTU(Wrk_MOoS);
   // If a Maintenance Out of Service command is received, and if Maintenance Out of Service
   // is configured to exist, place Out of Service (acquire MOoS).
   11: XIC(MCmd_OoS)OTU(MCmd_OoS)XIC(Cfg_HasMOoS)OTL(Wrk_MOoS);
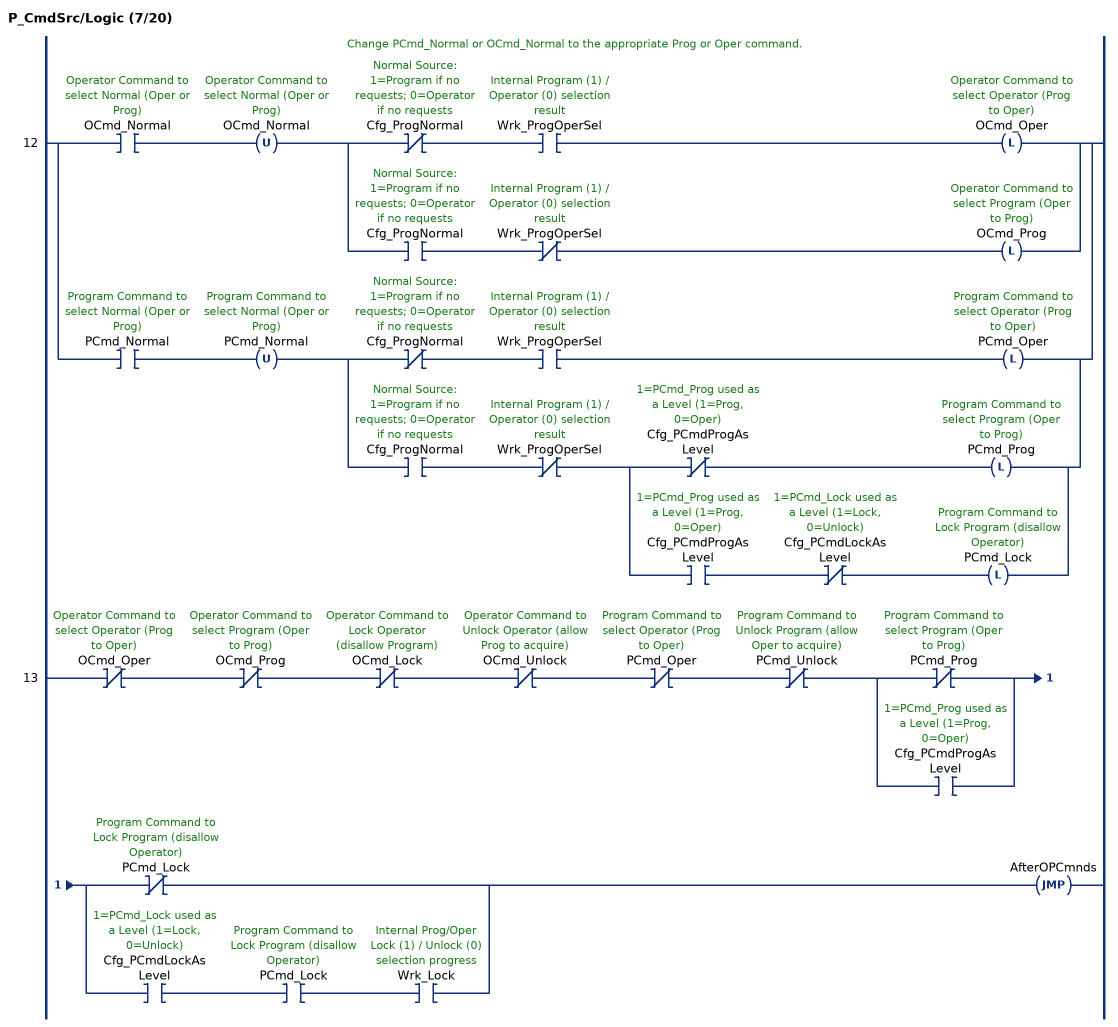
   // Change PCmd_Normal or OCmd_Normal to the appropriate Prog or Oper command.
   12: [XIC(OCmd_Normal) OTU(OCmd_Normal) [XIO(Cfg_ProgNormal) XIC(Wrk_ProgOperSel) OTL(OCmd_Oper) ,XIC(Cfg_ProgNormal) XIO(Wrk_ProgOperSel) OTL(OCmd_Prog) ] ,XIC(PCmd_Normal) OTU(PCmd_Normal) [XIO(Cfg_ProgNormal) XIC(Wrk_ProgOperSel) OTL(PCmd_Oper) ,XIC(Cfg_ProgNormal) XIO(Wrk_ProgOperSel) [XIO(Cfg_PCmdProgAsLevel) OTL(PCmd_Prog) ,XIC(Cfg_PCmdProgAsLevel) XIO(Cfg_PCmdLockAsLevel) OTL(PCmd_Lock) ] ] ];
   13: XIO(OCmd_Oper)XIO(OCmd_Prog)XIO(OCmd_Lock)XIO(OCmd_Unlock)XIO(PCmd_Oper)XIO(PCmd_Unlock)[XIO(PCmd_Prog) ,XIC(Cfg_PCmdProgAsLevel) ][XIO(PCmd_Lock) ,XIC(Cfg_PCmdLockAsLevel) XIC(PCmd_Lock) XIC(Wrk_Lock) ]JMP(AfterOPCmnds);
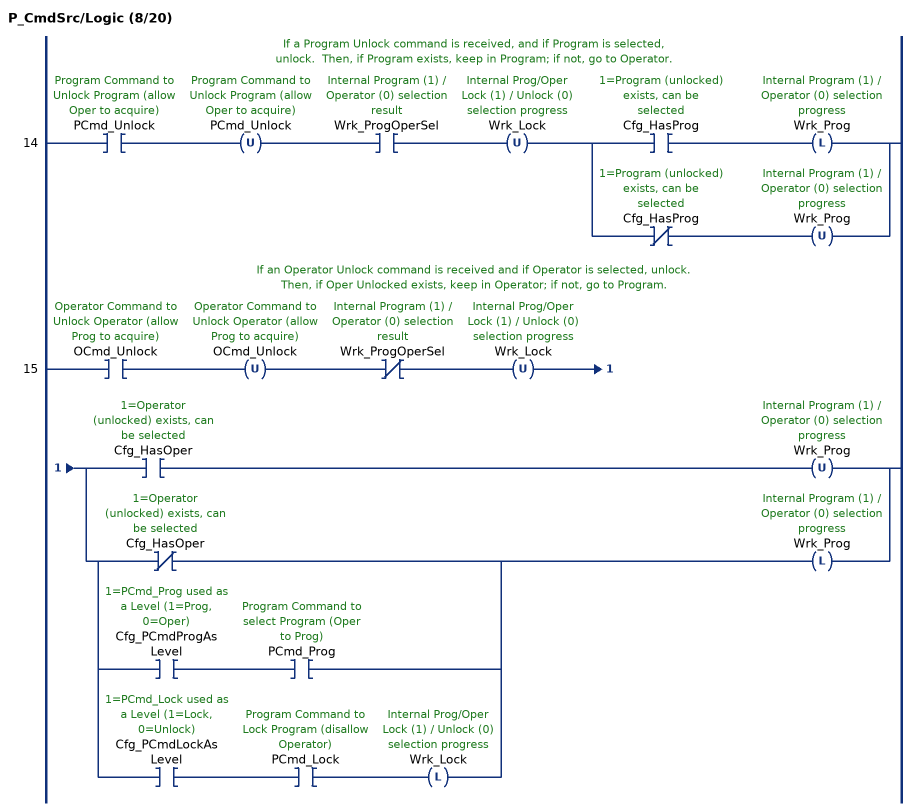
   // If a Program Unlock command is received, and if Program is selected,
   // unlock.  Then, if Program exists, keep in Program; if not, go to Operator.
   14: XIC(PCmd_Unlock)OTU(PCmd_Unlock)XIC(Wrk_ProgOperSel)OTU(Wrk_Lock)[XIC(Cfg_HasProg) OTL(Wrk_Prog) ,XIO(Cfg_HasProg) OTU(Wrk_Prog) ];
   // If an Operator Unlock command is received and if Operator is selected, unlock.
   // Then, if Oper Unlocked exists, keep in Operator; if not, go to Program.
   15: XIC(OCmd_Unlock)OTU(OCmd_Unlock)XIO(Wrk_ProgOperSel)OTU(Wrk_Lock)[XIC(Cfg_HasOper) OTU(Wrk_Prog) ,[XIO(Cfg_HasOper) ,XIC(Cfg_PCmdProgAsLevel) XIC(PCmd_Prog) ,XIC(Cfg_PCmdLockAsLevel) XIC(PCmd_Lock) OTL(Wrk_Lock) ] OTL(Wrk_Prog) ];
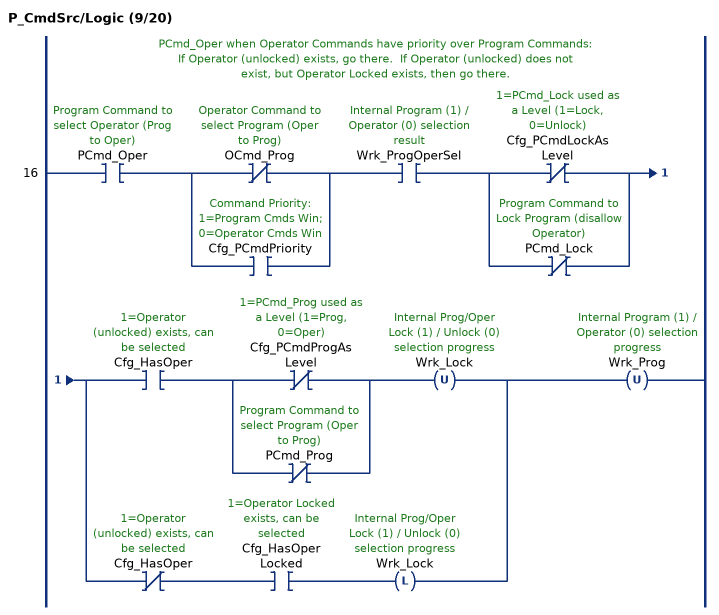
   // PCmd_Oper when Operator Commands have priority over Program Commands:
   // If Operator (unlocked) exists, go there.  If Operator (unlocked) does not
   // exist, but Operator Locked exists, then go there.
   16: XIC(PCmd_Oper)[XIO(OCmd_Prog) ,XIC(Cfg_PCmdPriority) ]XIC(Wrk_ProgOperSel)[XIO(Cfg_PCmdLockAsLevel) ,XIO(PCmd_Lock) ][XIC(Cfg_HasOper) [XIO(Cfg_PCmdProgAsLevel) ,XIO(PCmd_Prog) ] OTU(Wrk_Lock) ,XIO(Cfg_HasOper) XIC(Cfg_HasOperLocked) OTL(Wrk_Lock) ]OTU(Wrk_Prog);
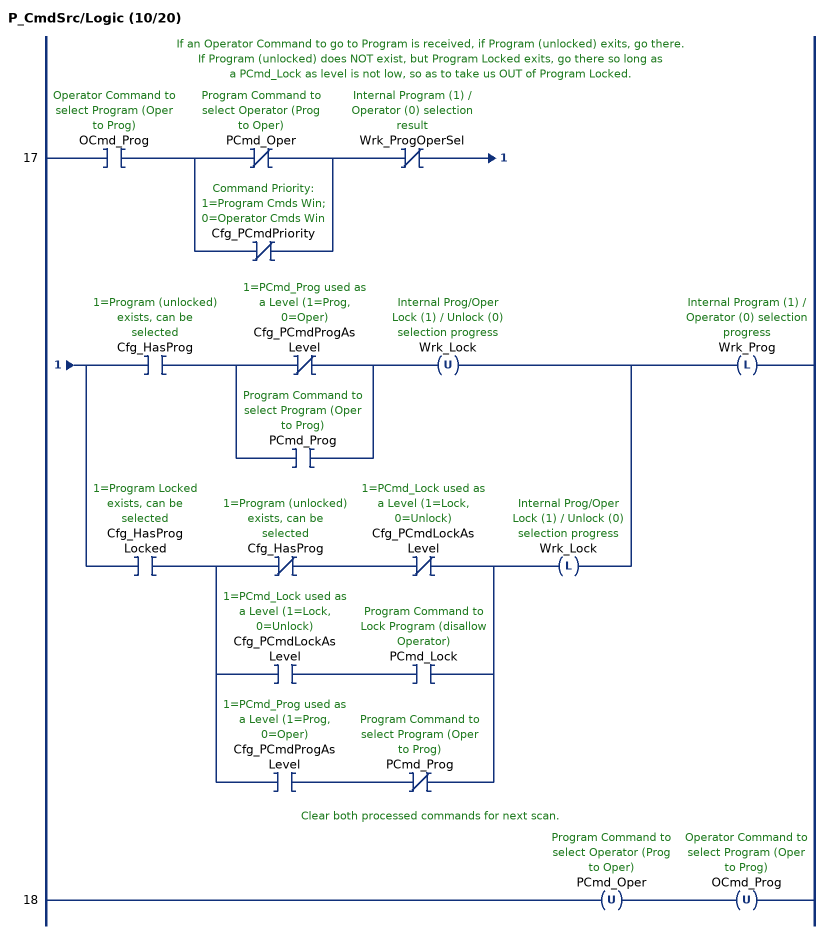
   // If an Operator Command to go to Program is received, if Program (unlocked) exits, go there.
   // If Program (unlocked) does NOT exist, but Program Locked exits, go there so long as
   // a PCmd_Lock as level is not low, so as to take us OUT of Program Locked.
   17: XIC(OCmd_Prog)[XIO(PCmd_Oper) ,XIO(Cfg_PCmdPriority) ]XIO(Wrk_ProgOperSel)[XIC(Cfg_HasProg) [XIO(Cfg_PCmdProgAsLevel) ,XIC(PCmd_Prog) ] OTU(Wrk_Lock) ,XIC(Cfg_HasProgLocked) [XIO(Cfg_HasProg) XIO(Cfg_PCmdLockAsLevel) ,XIC(Cfg_PCmdLockAsLevel) XIC(PCmd_Lock) ,XIC(Cfg_PCmdProgAsLevel) XIO(PCmd_Prog) ] OTL(Wrk_Lock) ]OTL(Wrk_Prog);
   // Clear both processed commands for next scan.
   18: OTU(PCmd_Oper)OTU(OCmd_Prog);
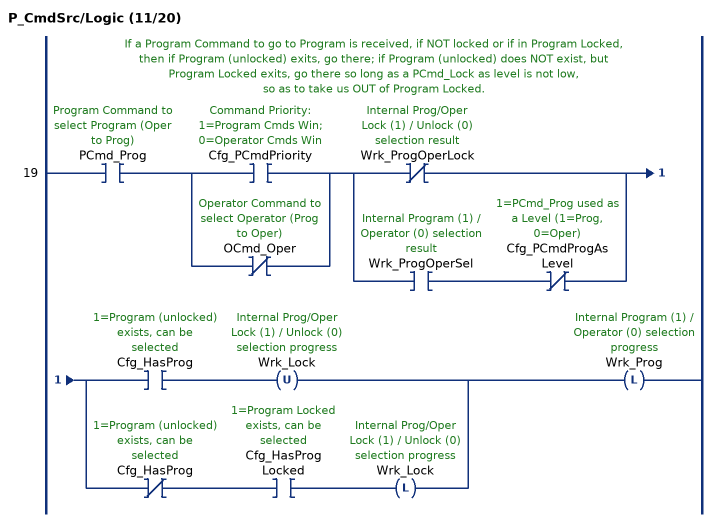
   // If a Program Command to go to Program is received, if NOT locked or if in Program Locked,
   // then if Program (unlocked) exits, go there; if Program (unlocked) does NOT exist, but
   // Program Locked exits, go there so long as a PCmd_Lock as level is not low,
   // so as to take us OUT of Program Locked.
   19: XIC(PCmd_Prog)[XIC(Cfg_PCmdPriority) ,XIO(OCmd_Oper) ][XIO(Wrk_ProgOperLock) ,XIC(Wrk_ProgOperSel) XIO(Cfg_PCmdProgAsLevel) ][XIC(Cfg_HasProg) OTU(Wrk_Lock) ,XIO(Cfg_HasProg) XIC(Cfg_HasProgLocked) OTL(Wrk_Lock) ]OTL(Wrk_Prog);
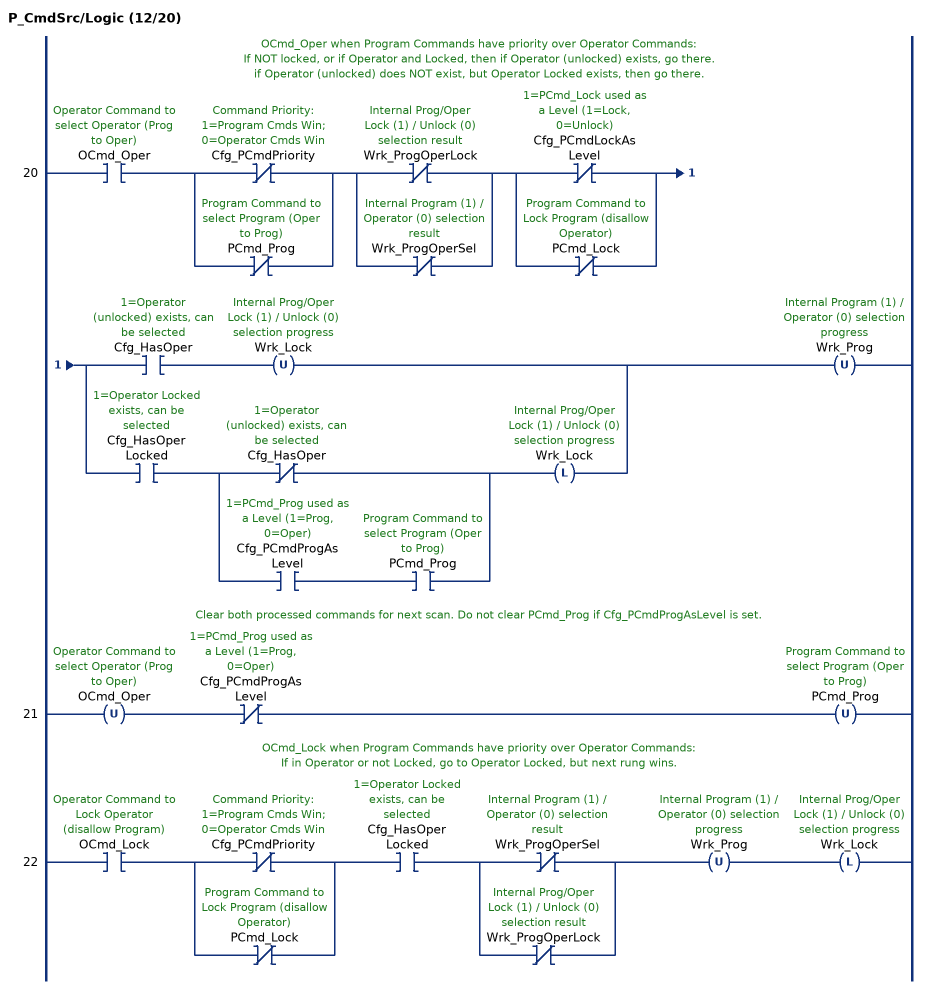
   // OCmd_Oper when Program Commands have priority over Operator Commands:
   // If NOT locked, or if Operator and Locked, then if Operator (unlocked) exists, go there.
   // if Operator (unlocked) does NOT exist, but Operator Locked exists, then go there.
   20: XIC(OCmd_Oper)[XIO(Cfg_PCmdPriority) ,XIO(PCmd_Prog) ][XIO(Wrk_ProgOperLock) ,XIO(Wrk_ProgOperSel) ][XIO(Cfg_PCmdLockAsLevel) ,XIO(PCmd_Lock) ][XIC(Cfg_HasOper) OTU(Wrk_Lock) ,XIC(Cfg_HasOperLocked) [XIO(Cfg_HasOper) ,XIC(Cfg_PCmdProgAsLevel) XIC(PCmd_Prog) ] OTL(Wrk_Lock) ]OTU(Wrk_Prog);
   // Clear both processed commands for next scan. Do not clear PCmd_Prog if Cfg_PCmdProgAsLevel is set.
   21: OTU(OCmd_Oper)XIO(Cfg_PCmdProgAsLevel)OTU(PCmd_Prog);
   // OCmd_Lock when Program Commands have priority over Operator Commands:
   // If in Operator or not Locked, go to Operator Locked, but next rung wins.
   22: XIC(OCmd_Lock)[XIO(Cfg_PCmdPriority) ,XIO(PCmd_Lock) ]XIC(Cfg_HasOperLocked)[XIO(Wrk_ProgOperSel) ,XIO(Wrk_ProgOperLock) ]OTU(Wrk_Prog)OTL(Wrk_Lock);
